// Mitsubishi GX Works2 project: Main_plc_id_1   PLC: FX3U/FX3UC

PROGRAM MAIN
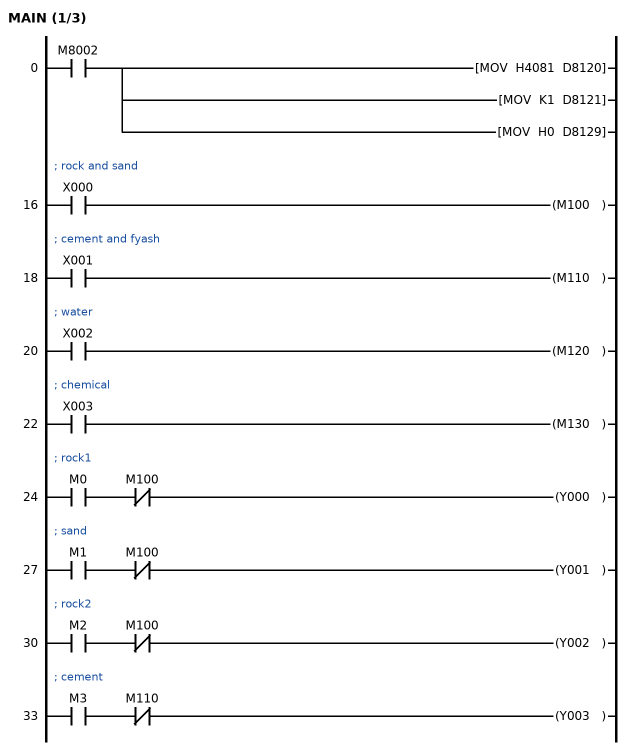
0     LD      M8002
      MOV     H4081 D8120
      MOV     K1 D8121
      MOV     H0 D8129
; rock and sand
16    LD      X000
      OUT     M100
; cement and fyash
18    LD      X001
      OUT     M110
; water
20    LD      X002
      OUT     M120
; chemical
22    LD      X003
      OUT     M130
; rock1
24    LD      M0
      ANI     M100
      OUT     Y000
; sand
27    LD      M1
      ANI     M100
      OUT     Y001
; rock2
30    LD      M2
      ANI     M100
      OUT     Y002
; cement
33    LD      M3
      ANI     M110
      OUT     Y003
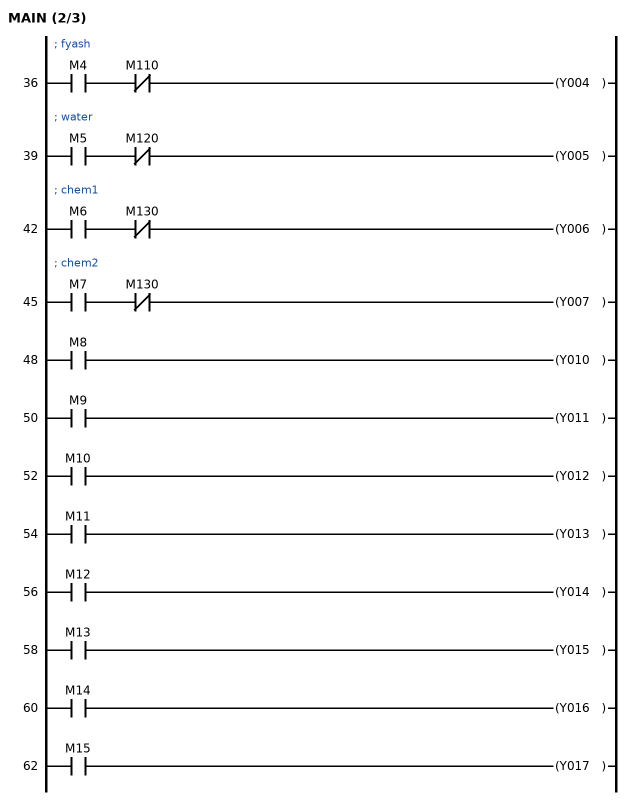
; fyash
36    LD      M4
      ANI     M110
      OUT     Y004
; water
39    LD      M5
      ANI     M120
      OUT     Y005
; chem1
42    LD      M6
      ANI     M130
      OUT     Y006
; chem2
45    LD      M7
      ANI     M130
      OUT     Y007
48    LD      M8
      OUT     Y010
50    LD      M9
      OUT     Y011
52    LD      M10
      OUT     Y012
54    LD      M11
      OUT     Y013
56    LD      M12
      OUT     Y014
58    LD      M13
      OUT     Y015
60    LD      M14
      OUT     Y016
62    LD      M15
      OUT     Y017
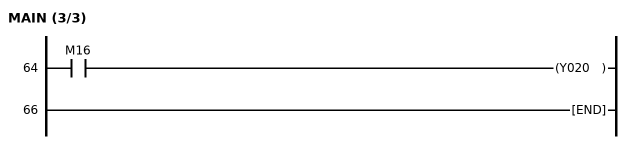
64    LD      M16
      OUT     Y020
66    END
END_PROGRAM
